// TwinCAT 3 PLC project PID_poging_2
// ProgramVersion: 3.1.4023.0
// libraries:
//   Tc2_ControllerToolbox, * (Beckhoff Automation GmbH)
//   Tc2_Standard, * (Beckhoff Automation GmbH)
//   Tc2_System, * (Beckhoff Automation GmbH)
//   Tc3_Module, * (Beckhoff Automation GmbH)
// project tree:
//   DUTs/ eModeTemperatureControl.TcDUT
//   GVLs/ GVL.TcGVL
//   / PlcTask.TcTTO
//   POUs/ FB_FruitTemperatureControl.TcPOU, MAIN.TcPOU

CONFIGURATION PID_poging_2
    RESOURCE PLC ON TwinCAT3
        TASK PlcTask(INTERVAL := T#1000ms, PRIORITY := 20);
        PROGRAM MAIN WITH PlcTask : MAIN;
    END_RESOURCE
END_CONFIGURATION

// ---- DUTs/eModeTemperatureControl.TcDUT
{attribute 'qualified_only'}
{attribute 'strict'}
TYPE eModeTemperatureControl :
(
	Normal := 0,
	Measure := 1,
	Control := 2
	//Alarm := 3 Deze bestaat niet want de input gaat dat overwriten
);
END_TYPE

// ---- GVLs/GVL.TcGVL
{attribute 'qualified_only'}
VAR_GLOBAL
	eTestMode : eModeTemperatureControl := eModeTemperatureControl.Normal; //Control mode
	fTestTsetOut : LREAL; //Calculated Tset
	fTestTthermostatOut : LREAL; //Adjsuted thermostat temperature
	fTestTthermostat : LREAL := -0.9; //input thermostat
	fTestTfruitRef : LREAL := -1;	//Reference temeprature
	fTestTfruit : LREAL := -0.75; //Fruit temperature
	bTestReset : BOOL; //Reset button
	// Control mode text
	sTestStateText : STRING (255);
	bRelay : BOOL; //output relay
	
	
	fTestKp : LREAL := 15;
	tTestKi : LREAL := 0.0136;
	tTestKt : LREAL := 0.0368;
	
	//outputs
	//Variables for checking the graph
	fTestUvoorSat : LREAL;
	fTestUerrorSat : LREAL;
	fTestUantiWind : LREAL;
	
END_VAR

// ---- POUs/MAIN.TcPOU
PROGRAM MAIN
VAR
	FB_TEST : FB_FruitTemperatureControl;
END_VAR

FB_TEST(//Input
		eControlMode := GVL.eTestMode,
		fTfruitRef := GVL.fTestTfruitRef,
		fTthermostat := GVL.fTestTthermostat,
		fTfruit := GVL.fTestTfruit,
		fKp := GVL.fTestKp,
		fKi := GVL.tTestKi,
		fKt := GVL.tTestKt,
		bReset := GVL.bTestReset,
		
		//Output
		fTthermostatOut => GVL.fTestTthermostatOut,
		sStateText => GVL.sTestStateText,
		bRelay => GVL.bRelay,
		
		//Test output
		fTestUantiWind => GVL.fTestUantiWind,
		fTestUerrorSat => GVL.fTestUerrorSat,
		fTestUvoorSat => GVL.fTestUvoorSat,
		fTestTsetOut => GVL.fTestTsetOut);

END_PROGRAM

// ---- POUs/FB_FruitTemperatureControl.TcPOU
FUNCTION_BLOCK FB_FruitTemperatureControl
VAR_INPUT
	fTfruitRef : LREAL;
	fTthermostat : LREAL; //AI Adres Thermostat
	fTfruit : LREAL; //AI Adress fruit temperature sensor
	
	fKp : LREAL;
	fKi : LREAL;
	fKt : LREAL;
	
	eControlMode : eModeTemperatureControl; //0 = Normal, 1 = Measure, 2 = Control
	bReset : BOOL; //Rising edge needed
END_VAR
VAR_OUTPUT
	fTthermostatOut : LREAL; //AQ Adres Thermostat out
	sStateText : STRING(255);
	bRelay : BOOL; //DQ relay
	
	fTestUvoorSat : LREAL; //Temporary output variables for graph 
	fTestUerrorSat : LREAL; //Temporary output variables for graph 
	fTestUantiWind : LREAL; //Temporary output variables for graph 
	fTestTsetOut : LREAL; //Temporary output variables for graph 
	
END_VAR
VAR
	tTi : TIME;
	tTt : TIME;
	//PI
	FB_PI : FB_CTRL_PI;
	ParamsPi : ST_CTRL_PI_PARAMS;
	eErrorIdPI : E_CTRL_ERRORCODES;
	bErrorPI : BOOL;
	//I
	FB_I : FB_CTRL_I;
	ParamsI : ST_CTRL_I_PARAMS;
	eErrorIdI : E_CTRL_ERRORCODES;
	bErrorI	 : BOOL;
	//Limiter
	FB_LIMIT : FB_CTRL_LIMITER;
	ParamsLimiter : ST_CTRL_LIMITER_PARAMS;
	eErrorIdLimiter : E_CTRL_ERRORCODES;
	bErrorLimiter	 : BOOL;
	fMinTset : LREAL;
	fMaxTset : LREAL;
	tCycleTime : TIME := T#1000MS; //Sampling time = 1s

	fTfruitZero : LREAL;
	fTsetZero : LREAL;
	bRunOnce : BOOL := TRUE;
	bSafety : BOOL := TRUE;
	rTrigger : R_TRIG;
	
	//controller output variables
	fUafterSat: LREAL;
	fUerrorSat: LREAL; 
	fUvoorSat: LREAL;
	fUantiWind: LREAL := 0;
	fUpi: LREAL;
	fTsetOut : LREAL;
	//Timer Tset =< -2°C
	bTimerAtMinus2 : BOOL := FALSE;
	tMaxTimeMinus2 : TIME := T#56000S; //15h33min20s
	bTimerAtMinus2Out : BOOL;
	TimerAtMinus2 : TON;
	tElapsedTimeAtMinus2 : TIME;
	
	//Timer Tset > -2°C
	bTimerAboveMinus2 : BOOL := FALSE;
	tMinTimeAboveMinus2 : TIME := T#1800S; //30min
	bTimerAboveMinus2Out : BOOL;
	TimerAboveMinus2 : TON;
	tElapsedTimeAboveMinus2 : TIME;
	bRtrigOut: BOOL;
END_VAR


//Integral gain to integral time
tTi := LREAL_TO_TIME((fKp/fKi)*1000);
tTt := LREAL_TO_TIME((1/fKt)*1000);	
//******************************************************************************//
IF (eControlMode = 2 AND bSafety = TRUE) THEN //Control mode
	IF bRunOnce THEN
		fTfruitZero := fTfruit; //Important that the cold store is running for a few days with Tset = TfruitRef
		fTsetZero := fTfruitRef;
		bRunOnce := FALSE;
	END_IF
	
	//PI blok
	ParamsPi.fKp := fKp;
	ParamsPi.tTn := tTi;
	ParamsPi.fOutMaxLimit := 1E38;
	ParamsPi.fOutMinLimit := -1E38;
	ParamsPi.tCtrlCycleTime := tCycleTime;
	ParamsPi.tTaskCycleTime:= tCycleTime;
	ParamsPi.bARWOnIPartOnly := TRUE;
	
	FB_PI(	fSetpointValue		:= fTfruitRef-fTfruitZero,
			fActualValue		:= fTfruit-fTfruitZero ,
			fManSyncValue	:= 0,
			bSync				:= FALSE,
			eMode				:= E_CTRL_MODE.eCTRL_MODE_ACTIVE,
			bHold				:= FALSE,
			stParams			:= ParamsPi,
			fOut				=> fUpi,
			bARWactive		=> ,
			eErrorId			=> eErrorIdPI,
			bError				=> bErrorPI
				);
	fUvoorSat := fUpi+fUantiWind;
		fTestUvoorSat:=fUvoorSat; 	//Test variabels
	//Limiter
	fMinTset := -1;
	fMaxTset := 3+fTfruitRef;
	
	
	ParamsLimiter.fMaxOutput := fMaxTset;
	ParamsLimiter.fMinOutput := fMinTset;
	ParamsLimiter.tCtrlCycleTime := tCycleTime;
	ParamsLimiter.tTaskCycleTime := tCycleTime;
	
	FB_LIMIT (	fIn					:= fUvoorSat,
			  	stParams			:= ParamsLimiter,
				fOut				=> fUafterSat,
				eErrorId			=> eErrorIdLimiter,
				bError				=> bErrorLimiter);
	
	//I blok
	ParamsI.fOutMaxLimit := 1E38;
	ParamsI.fOutMinLimit := -1E38;
	ParamsI.tCtrlCycleTime := tCycleTime;
	ParamsI.tTaskCycleTime := tCycleTime;
	ParamsI.tTi := tTt;
	
		fTestUerrorSat := fUerrorSat; 	//Test variabels
	fUerrorSat := fUafterSat-fUvoorSat;					
	FB_I(	fIn					:= fUerrorSat,
			eMode				:= E_CTRL_MODE.eCTRL_MODE_ACTIVE,
			stParams			:= ParamsI,
			fOut				=> fUantiWind,
			eErrorId			=> eErrorIdI,
			bError				=> bErrorI);
	fTestUantiWind := fUantiWind; 	//Test variabels
	//TsetOut to TthermostatOut
	fTsetOut := fUafterSat + fTsetZero;
	fTthermostatOut := fTthermostat + (fTsetOut-fTsetZero);
	
		fTestTsetOut := fTsetOut; 	//Test variabels
		GVL.fTestTthermostatOut := fTthermostatOut;	//Test variabels
	//-2°C timer
	IF(fTsetOut > -2) THEN
		bTimerAboveMinus2 := TRUE;
	ELSE
		bTimerAboveMinus2 := FALSE;
	END_IF
	//*********************************************************************//
	TimerAboveMinus2(IN := bTimerAboveMinus2,
					PT := tMinTimeAboveMinus2,
					Q => bTimerAboveMinus2Out,
					ET => tElapsedTimeAboveMinus2);
 	IF(bTimerAboveMinus2Out = TRUE) THEN //We are safe
		bTimerAboveMinus2 := FALSE;
		TimerAboveMinus2(IN := bTimerAboveMinus2,
			PT := tMinTimeAboveMinus2,
			Q => bTimerAboveMinus2Out,
			ET => tElapsedTimeAboveMinus2);
					
		bTimerAtMinus2 := FALSE;
		TimerAtMinus2(IN := bTimerAtMinus2,
			PT := tMaxTimeMinus2,
			Q => bTimerAtMinus2Out,
			ET => tElapsedTimeAtMinus2);	
			
	END_IF
	 
	IF (fTsetOut <= -2 AND NOT(bTimerAboveMinus2Out))THEN
		bTimerAtMinus2 := TRUE;	
	END_IF
	TimerAtMinus2(IN := bTimerAtMinus2,
		PT := tMaxTimeMinus2,
		Q => bTimerAtMinus2Out,
		ET => tElapsedTimeAtMinus2);
	IF(bTimerAtMinus2Out) THEN //To long at -2
		bSafety := FALSE;
	END_IF
	
	sStateText := 'PI temperature control is running';
	bRelay := TRUE;
//******************************************************************************//
ELSE
	IF(eControlMode = 1 AND bSafety = TRUE)THEN //Measurement mode
		bRunOnce := TRUE;
		
		//Resetting PI, I and TON
		bTimerAtMinus2 := FALSE;
		TimerAtMinus2(IN := bTimerAtMinus2,
			PT := tMaxTimeMinus2,
			Q => bTimerAtMinus2Out,
			ET => tElapsedTimeAtMinus2);
		
		bTimerAboveMinus2 := FALSE; 
		TimerAboveMinus2(IN := bTimerAboveMinus2,
			PT := tMinTimeAboveMinus2,
			Q => bTimerAboveMinus2Out,
			ET => tElapsedTimeAboveMinus2);

		FB_PI(fSetpointValue		:= fTfruitRef-fTfruitZero,
			fActualValue		:= fTfruit-fTfruitZero ,
			fManSyncValue	:= 0,
			bSync				:= FALSE,
			eMode				:= E_CTRL_MODE.eCTRL_MODE_RESET,
			bHold				:= FALSE,
			stParams			:= ParamsPi,
			fOut				=> fUpi,
			bARWactive		=> ,
			eErrorId			=> eErrorIdPI,
			bError				=> bErrorPI);
		FB_I(fIn				:= fUerrorSat,
			eMode				:= E_CTRL_MODE.eCTRL_MODE_RESET,
			stParams			:= ParamsI,
			fOut				=> fUantiWind,
			eErrorId			=> eErrorIdI,
			bError				=> bErrorI);
		fTthermostatOut := fTthermostat;
		sStateText := 'Normal control and collecting data';
		bRelay := TRUE;

		//Data measurement algoritm;
	 	
	END_IF
//******************************************************************************//	
	IF (eControlMode = 0 AND bSafety = TRUE) THEN //Normal mode
		bRunOnce := TRUE;
		
		//Resetting PI, I and TON
		bTimerAtMinus2 := FALSE;
		TimerAtMinus2(IN := bTimerAtMinus2,
			PT := tMaxTimeMinus2,
			Q => bTimerAtMinus2Out,
			ET => tElapsedTimeAtMinus2);
		
		bTimerAboveMinus2 := FALSE; 
		TimerAboveMinus2(IN := bTimerAboveMinus2,
			PT := tMinTimeAboveMinus2,
			Q => bTimerAboveMinus2Out,
			ET => tElapsedTimeAboveMinus2);
		
		FB_PI(fSetpointValue		:= fTfruitRef-fTfruitZero,
			fActualValue		:= fTfruit-fTfruitZero ,
			fManSyncValue	:= 0,
			bSync				:= FALSE,
			eMode				:= E_CTRL_MODE.eCTRL_MODE_RESET,
			bHold				:= FALSE,
			stParams			:= ParamsPi,
			fOut				=> fUpi,
			bARWactive		=> ,
			eErrorId			=> eErrorIdPI,
			bError				=> bErrorPI);
		FB_I(fIn				:= fUerrorSat,
			eMode				:= E_CTRL_MODE.eCTRL_MODE_RESET,
			stParams			:= ParamsI,
			fOut				=> fUantiWind,
			eErrorId			=> eErrorIdI,
			bError				=> bErrorI);
		
		fTthermostatOut := fTthermostat;
		sStateText := 'Normal control and NOT collecting data';
		bRelay := FALSE;
		
	END_IF
//******************************************************************************//	
	IF NOT bSafety THEN //Error state
		
		//Resetting PI, I and TON
		bRunOnce := TRUE;
		bTimerAtMinus2 := FALSE;
		TimerAtMinus2(IN := bTimerAtMinus2,
			PT := tMaxTimeMinus2,
			Q => bTimerAtMinus2Out,
			ET => tElapsedTimeAtMinus2);
		
		bTimerAboveMinus2 := FALSE; 
		TimerAboveMinus2(IN := bTimerAboveMinus2,
			PT := tMinTimeAboveMinus2,
			Q => bTimerAboveMinus2Out,
			ET => tElapsedTimeAboveMinus2);

		
		FB_PI(fSetpointValue		:= fTfruitRef-fTfruitZero,
			fActualValue		:= fTfruit-fTfruitZero ,
			fManSyncValue	:= 0,
			bSync				:= FALSE,
			eMode				:= E_CTRL_MODE.eCTRL_MODE_RESET,
			bHold				:= FALSE,
			stParams			:= ParamsPi,
			fOut				=> fUpi,
			bARWactive		=> ,
			eErrorId			=> eErrorIdPI,
			bError				=> bErrorPI);
		FB_I(fIn				:= fUerrorSat,
			eMode				:= E_CTRL_MODE.eCTRL_MODE_RESET,
			stParams			:= ParamsI,
			fOut				=> fUantiWind,
			eErrorId			=> eErrorIdI,
			bError				=> bErrorI);
			
		//Reset button with rising edge
		rTrigger(CLK:=bReset,
					Q => bRtrigOut);
		IF(bRtrigOut = TRUE) THEN
			bSafety := TRUE;
		END_IF
		
		sStateText := 'Error mode, settemperature remained to long at -2°C. Press reset in order to acces other control modes.
						Normal operation without data collecting currently active';
		bRelay := FALSE;
		fTthermostatOut := fTthermostat;
	END_IF
END_IF

END_FUNCTION_BLOCK
